FUNCTION_BLOCK IMG_BOOL (* Boolean Input Checkbox with Label and Image *)
  (* Standard: 61499-1; Function: HMI; Type: BOOL input; Description: Checkbox with Image *)
  (* Version 0.0, 2006-07-03, JHC, Holobloc Inc, Adapted from IN_BOOL. *)
  (* Compiler header: package fb.rt.hmi; import javax.swing.*; *)
  (* Compiler classdef: public class IMG_BOOL extends IN_BOOL *)
  (* Compiler Java IBM VisualAge 3.0 *)
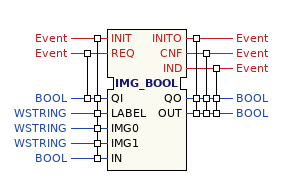
  EVENT_INPUT
    INIT WITH QI, LABEL, IN, IMG0, IMG1; (* Initialization *)
    REQ WITH QI; (* Request *)
  END_EVENT
  EVENT_OUTPUT
    INITO WITH QO, OUT; (* Initialization Confirm *)
    CNF WITH QO, OUT; (* Service Confirmation *)
    IND WITH QO, OUT; (* User clicked Checkbox *)
  END_EVENT
  VAR_INPUT
    QI : BOOL := true; (* Event qualifier *)
    LABEL : WSTRING; (* Label *)
    IMG0 : WSTRING; (* Image location, e.g., "images/Stop16.gif", for unselected (0) state *)
    IMG1 : WSTRING; (* Image location, e.g., "images/Stop24.gif", for selected (1) state *)
    IN : BOOL; (* Initial value *)
  END_VAR
  VAR_OUTPUT
    QO : BOOL; (* Event qualifier *)
    OUT : BOOL; (* Output data *)
  END_VAR
  SERVICE IN_BOOL/Checkbox
    SEQUENCE normal_initialization
      IN_BOOL.INIT+(LABEL,IMG0,IMG1,IN) -> Checkbox.setLabel(LABEL) -> Checkbox.setIcon(IMG0) -> Checkbox.setSelectedIcon(IMG1) -> Checkbox.setState(IN) -> IN_BOOL.INITO+();
    END_SEQUENCE
    SEQUENCE initialization_inhibited
      IN_BOOL.INIT-() -> IN_BOOL.INITO-();
    END_SEQUENCE
    SEQUENCE data_read
      IN_BOOL.REQ+() -> Checkbox.getState() -> IN_BOOL.CNF+(OUT);
    END_SEQUENCE
    SEQUENCE user_input
      Checkbox.itemStateChanged() -> IN_BOOL.IND+(OUT);
    END_SEQUENCE
  END_SERVICE
END_FUNCTION_BLOCK
